// Mitsubishi GX Works2 project: pr1   PLC: Q03UDV

PROGRAM MAIN
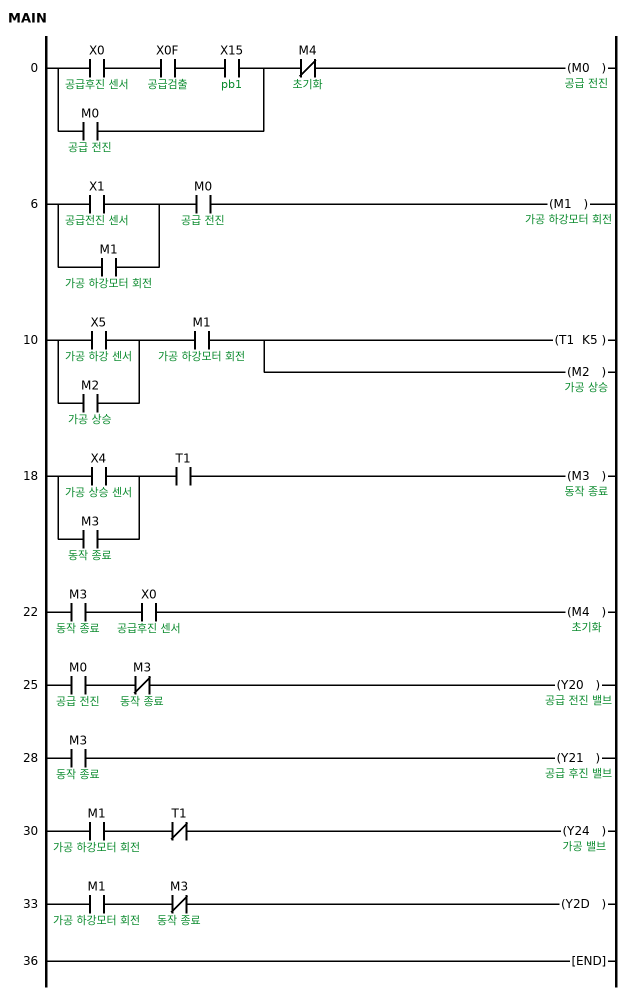
0     LD      X0  ; 공급후진 센서
      AND     X0F  ; 공급검출
      AND     X15  ; pb1
      OR      M0  ; 공급 전진
      ANI     M4  ; 초기화
      OUT     M0  ; 공급 전진
6     LD      X1  ; 공급전진 센서
      OR      M1  ; 가공 하강모터 회전
      AND     M0  ; 공급 전진
      OUT     M1  ; 가공 하강모터 회전
10    LD      X5  ; 가공 하강 센서
      OR      M2  ; 가공 상승
      AND     M1  ; 가공 하강모터 회전
      OUT     T1 K5
      OUT     M2  ; 가공 상승
18    LD      X4  ; 가공 상승 센서
      OR      M3  ; 동작 종료
      AND     T1
      OUT     M3  ; 동작 종료
22    LD      M3  ; 동작 종료
      AND     X0  ; 공급후진 센서
      OUT     M4  ; 초기화
25    LD      M0  ; 공급 전진
      ANI     M3  ; 동작 종료
      OUT     Y20  ; 공급 전진 밸브
28    LD      M3  ; 동작 종료
      OUT     Y21  ; 공급 후진 밸브
30    LD      M1  ; 가공 하강모터 회전
      ANI     T1
      OUT     Y24  ; 가공 밸브
33    LD      M1  ; 가공 하강모터 회전
      ANI     M3  ; 동작 종료
      OUT     Y2D
36    END
END_PROGRAM

// device comments not shown above
X6  ; 가공 하강 센서
